# B&R Automation Studio project DivDiag (part 2)

### DivertRepo.mpreportcore - PC/mappServices/DivertRepo.mpreportcore
```
Element gOffsetsReport (Type=mpreportcore)
  MpReport:
    Settings:
      ResourceDeviceName = 
      LanguageDependent:
        [0]:
          Language = en
          Font = 1
    PageLayouts:
      [0]:
        Name = Default
        PageFormat = 1
    Styles:
      Text:
        [0]:
          Name = Default
        [1]:
          Name = Title
          Style = 1
          Size = 14
        [2]:
          Name = Header
          Size = 12
        [3]:
          Name = Section
          Style = 2
          Size = 12
      Table:
        [0]:
          Name = Default
      Line:
        [0]:
          Name = Default
      Chart:
        PieChart:
          [0]:
            Name = Default
        LineChart:
          [0]:
            Name = Default
        BarChart:
          [0]:
            Name = Default
    Tables:
      [0]:
        Name = Divert1
        TableStyle = Default
        TextStyle = Default
        [0]:
          [0] = TextId
            Source = 
            Width = 40
          [1] = TextId
            Source = Segment 1
          [2] = TextId
            Source = Segment 2
        [1]:
          [0] = TextId
            Source = Name
            Width = 40
          [1] = ValueId
            Value:
              ProcessVariable = ::Maint:TestResults[0].Seg1Name
          [2] = ValueId
            Value:
              ProcessVariable = ::Maint:TestResults[0].Seg2Name
        [2]:
          [0] = TextId
            Source = Type
            Width = 40
          [1] = ValueId
            Value:
              ProcessVariable = ::Maint:TestResults[0].Seg1Type
          [2] = ValueId
            Value:
              ProcessVariable = ::Maint:TestResults[0].Seg2Type
        [3]:
          [0] = TextId
            Source = Relative to start of segment
            Width = 40
          [1] = ValueId
            Value:
              ProcessVariable = ::Maint:TestResults[0].Seg1PosRelToStart
          [2] = ValueId
            Value:
              ProcessVariable = ::Maint:TestResults[0].Seg2PosRelToStart
        [4]:
          [0] = TextId
            Source = Relative to end of segment
            Width = 40
          [1] = ValueId
            Value:
              ProcessVariable = ::Maint:TestResults[0].Seg1PosRelToEnd
          [2] = ValueId
            Value:
              ProcessVariable = ::Maint:TestResults[0].Seg2PosRelToEnd
        [5]:
          [0] = TextId
            Source = Measured Configuration Mismatch
            Width = 40
          [1] = ValueId
            Value:
              ProcessVariable = ::Maint:TestResults[0].Deviation
            Width = 50
            HorizontalAlign = 1
      [1]:
        Name = Divert2
        TableStyle = Default
        TextStyle = Default
        [0]:
          [0] = TextId
            Source = 
            Width = 40
          [1] = TextId
            Source = Segment 1
          [2] = TextId
            Source = Segment 2
        [1]:
          [0] = TextId
            Source = Name
            Width = 40
          [1] = ValueId
            Value:
              ProcessVariable = ::Maint:TestResults[1].Seg1Name
          [2] = ValueId
            Value:
              ProcessVariable = ::Maint:TestResults[1].Seg2Name
        [2]:
          [0] = TextId
            Source = Type
            Width = 40
          [1] = ValueId
            Value:
              ProcessVariable = ::Maint:TestResults[1].Seg1Type
          [2] = ValueId
            Value:
              ProcessVariable = ::Maint:TestResults[1].Seg2Type
        [3]:
          [0] = TextId
            Source = Relative to start of segment
            Width = 40
          [1] = ValueId
            Value:
              ProcessVariable = ::Maint:TestResults[1].Seg1PosRelToStart
          [2] = ValueId
            Value:
              ProcessVariable = ::Maint:TestResults[1].Seg2PosRelToStart
        [4]:
          [0] = TextId
            Source = Relative to end of segment
            Width = 40
          [1] = ValueId
            Value:
              ProcessVariable = ::Maint:TestResults[1].Seg1PosRelToEnd
          [2] = ValueId
            Value:
              ProcessVariable = ::Maint:TestResults[1].Seg2PosRelToEnd
        [5]:
          [0] = TextId
            Source = Measured Configuration Mismatch
            Width = 40
          [1] = ValueId
            Value:
              ProcessVariable = ::Maint:TestResults[1].Deviation
            Width = 50
            HorizontalAlign = 1
      [2]:
        Name = Divert3
        TableStyle = Default
        TextStyle = Default
        [0]:
          [0] = TextId
            Source = 
            Width = 40
          [1] = TextId
            Source = Segment 1
          [2] = TextId
            Source = Segment 2
        [1]:
          [0] = TextId
            Source = Name
            Width = 40
          [1] = ValueId
            Value:
              ProcessVariable = ::Maint:TestResults[2].Seg1Name
          [2] = ValueId
            Value:
              ProcessVariable = ::Maint:TestResults[2].Seg2Name
        [2]:
          [0] = TextId
            Source = Type
            Width = 40
          [1] = ValueId
            Value:
              ProcessVariable = ::Maint:TestResults[2].Seg1Type
          [2] = ValueId
            Value:
              ProcessVariable = ::Maint:TestResults[2].Seg2Type
        [3]:
          [0] = TextId
            Source = Relative to start of segment
            Width = 40
          [1] = ValueId
            Value:
              ProcessVariable = ::Maint:TestResults[2].Seg1PosRelToStart
          [2] = ValueId
            Value:
              ProcessVariable = ::Maint:TestResults[2].Seg2PosRelToStart
        [4]:
          [0] = TextId
            Source = Relative to end of segment
            Width = 40
          [1] = ValueId
            Value:
              ProcessVariable = ::Maint:TestResults[2].Seg1PosRelToEnd
          [2] = ValueId
            Value:
              ProcessVariable = ::Maint:TestResults[2].Seg2PosRelToEnd
        [5]:
          [0] = TextId
            Source = Measured Configuration Mismatch
            Width = 40
          [1] = ValueId
            Value:
              ProcessVariable = ::Maint:TestResults[2].Deviation
            Width = 50
            HorizontalAlign = 1
      [3]:
        Name = Divert4
        TableStyle = Default
        TextStyle = Default
        [0]:
          [0] = TextId
            Source = 
            Width = 40
          [1] = TextId
            Source = Segment 1
          [2] = TextId
            Source = Segment 2
        [1]:
          [0] = TextId
            Source = Name
            Width = 40
          [1] = ValueId
            Value:
              ProcessVariable = ::Maint:TestResults[3].Seg1Name
          [2] = ValueId
            Value:
              ProcessVariable = ::Maint:TestResults[3].Seg2Name
        [2]:
          [0] = TextId
            Source = Type
            Width = 40
          [1] = ValueId
            Value:
              ProcessVariable = ::Maint:TestResults[3].Seg1Type
          [2] = ValueId
            Value:
              ProcessVariable = ::Maint:TestResults[3].Seg2Type
        [3]:
          [0] = TextId
            Source = Relative to start of segment
            Width = 40
          [1] = ValueId
            Value:
              ProcessVariable = ::Maint:TestResults[3].Seg1PosRelToStart
          [2] = ValueId
            Value:
              ProcessVariable = ::Maint:TestResults[3].Seg2PosRelToStart
        [4]:
          [0] = TextId
            Source = Relative to end of segment
            Width = 40
          [1] = ValueId
            Value:
              ProcessVariable = ::Maint:TestResults[3].Seg1PosRelToEnd
          [2] = ValueId
            Value:
              ProcessVariable = ::Maint:TestResults[3].Seg2PosRelToEnd
        [5]:
          [0] = TextId
            Source = Measured Configuration Mismatch
            Width = 40
          [1] = ValueId
            Value:
              ProcessVariable = ::Maint:TestResults[3].Deviation
            Width = 50
            HorizontalAlign = 1
      [4]:
        Name = Divert5
        TableStyle = Default
        TextStyle = Default
        [0]:
          [0] = TextId
            Source = 
            Width = 40
          [1] = TextId
            Source = Segment 1
          [2] = TextId
            Source = Segment 2
        [1]:
          [0] = TextId
            Source = Name
            Width = 40
          [1] = ValueId
            Value:
              ProcessVariable = ::Maint:TestResults[4].Seg1Name
          [2] = ValueId
            Value:
              ProcessVariable = ::Maint:TestResults[4].Seg2Name
        [2]:
          [0] = TextId
            Source = Type
            Width = 40
          [1] = ValueId
            Value:
              ProcessVariable = ::Maint:TestResults[4].Seg1Type
          [2] = ValueId
            Value:
              ProcessVariable = ::Maint:TestResults[4].Seg2Type
        [3]:
          [0] = TextId
            Source = Relative to start of segment
            Width = 40
          [1] = ValueId
            Value:
              ProcessVariable = ::Maint:TestResults[4].Seg1PosRelToStart
          [2] = ValueId
            Value:
              ProcessVariable = ::Maint:TestResults[4].Seg2PosRelToStart
        [4]:
          [0] = TextId
            Source = Relative to end of segment
            Width = 40
          [1] = ValueId
            Value:
              ProcessVariable = ::Maint:TestResults[4].Seg1PosRelToEnd
          [2] = ValueId
            Value:
              ProcessVariable = ::Maint:TestResults[4].Seg2PosRelToEnd
        [5]:
          [0] = TextId
            Source = Measured Configuration Mismatch
            Width = 40
          [1] = ValueId
            Value:
              ProcessVariable = ::Maint:TestResults[4].Deviation
            Width = 50
            HorizontalAlign = 1
      [5]:
        Name = Divert6
        TableStyle = Default
        TextStyle = Default
        [0]:
          [0] = TextId
            Source = 
            Width = 40
          [1] = TextId
            Source = Segment 1
          [2] = TextId
            Source = Segment 2
        [1]:
          [0] = TextId
            Source = Name
            Width = 40
          [1] = ValueId
            Value:
              ProcessVariable = ::Maint:TestResults[5].Seg1Name
          [2] = ValueId
            Value:
              ProcessVariable = ::Maint:TestResults[5].Seg2Name
        [2]:
          [0] = TextId
            Source = Type
            Width = 40
          [1] = ValueId
            Value:
              ProcessVariable = ::Maint:TestResults[5].Seg1Type
          [2] = ValueId
            Value:
              ProcessVariable = ::Maint:TestResults[5].Seg2Type
        [3]:
          [0] = TextId
            Source = Relative to start of segment
            Width = 40
          [1] = ValueId
            Value:
              ProcessVariable = ::Maint:TestResults[5].Seg1PosRelToStart
          [2] = ValueId
            Value:
              ProcessVariable = ::Maint:TestResults[5].Seg2PosRelToStart
        [4]:
          [0] = TextId
            Source = Relative to end of segment
            Width = 40
          [1] = ValueId
            Value:
              ProcessVariable = ::Maint:TestResults[5].Seg1PosRelToEnd
          [2] = ValueId
            Value:
              ProcessVariable = ::Maint:TestResults[5].Seg2PosRelToEnd
        [5]:
          [0] = TextId
            Source = Measured Configuration Mismatch
            Width = 40
          [1] = ValueId
            Value:
              ProcessVariable = ::Maint:TestResults[5].Deviation
            Width = 50
            HorizontalAlign = 1
      [6]:
        Name = Divert7
        TableStyle = Default
        TextStyle = Default
        [0]:
          [0] = TextId
            Source = 
            Width = 40
          [1] = TextId
            Source = Segment 1
          [2] = TextId
            Source = Segment 2
        [1]:
          [0] = TextId
            Source = Name
            Width = 40
          [1] = ValueId
            Value:
              ProcessVariable = ::Maint:TestResults[6].Seg1Name
          [2] = ValueId
            Value:
              ProcessVariable = ::Maint:TestResults[6].Seg2Name
        [2]:
          [0] = TextId
            Source = Type
            Width = 40
          [1] = ValueId
            Value:
              ProcessVariable = ::Maint:TestResults[6].Seg1Type
          [2] = ValueId
            Value:
              ProcessVariable = ::Maint:TestResults[6].Seg2Type
        [3]:
          [0] = TextId
            Source = Relative to start of segment
            Width = 40
          [1] = ValueId
            Value:
              ProcessVariable = ::Maint:TestResults[6].Seg1PosRelToStart
          [2] = ValueId
            Value:
              ProcessVariable = ::Maint:TestResults[6].Seg2PosRelToStart
        [4]:
          [0] = TextId
            Source = Relative to end of segment
            Width = 40
          [1] = ValueId
            Value:
              ProcessVariable = ::Maint:TestResults[6].Seg1PosRelToEnd
          [2] = ValueId
            Value:
              ProcessVariable = ::Maint:TestResults[6].Seg2PosRelToEnd
        [5]:
          [0] = TextId
            Source = Measured Configuration Mismatch
            Width = 40
          [1] = ValueId
            Value:
              ProcessVariable = ::Maint:TestResults[6].Deviation
            Width = 50
            HorizontalAlign = 1
      [7]:
        Name = Divert8
        TableStyle = Default
        TextStyle = Default
        [0]:
          [0] = TextId
            Source = 
            Width = 40
          [1] = TextId
            Source = Segment 1
          [2] = TextId
            Source = Segment 2
        [1]:
          [0] = TextId
            Source = Name
            Width = 40
          [1] = ValueId
            Value:
              ProcessVariable = ::Maint:TestResults[7].Seg1Name
          [2] = ValueId
            Value:
              ProcessVariable = ::Maint:TestResults[7].Seg2Name
        [2]:
          [0] = TextId
            Source = Type
            Width = 40
          [1] = ValueId
            Value:
              ProcessVariable = ::Maint:TestResults[7].Seg1Type
          [2] = ValueId
            Value:
              ProcessVariable = ::Maint:TestResults[7].Seg2Type
        [3]:
          [0] = TextId
            Source = Relative to start of segment
            Width = 40
          [1] = ValueId
            Value:
              ProcessVariable = ::Maint:TestResults[7].Seg1PosRelToStart
          [2] = ValueId
            Value:
              ProcessVariable = ::Maint:TestResults[7].Seg2PosRelToStart
        [4]:
          [0] = TextId
            Source = Relative to end of segment
            Width = 40
          [1] = ValueId
            Value:
              ProcessVariable = ::Maint:TestResults[7].Seg1PosRelToEnd
          [2] = ValueId
            Value:
              ProcessVariable = ::Maint:TestResults[7].Seg2PosRelToEnd
        [5]:
          [0] = TextId
            Source = Measured Configuration Mismatch
            Width = 40
          [1] = ValueId
            Value:
              ProcessVariable = ::Maint:TestResults[7].Deviation
            Width = 50
            HorizontalAlign = 1
      [8]:
        Name = Divert9
        TableStyle = Default
        TextStyle = Default
        [0]:
          [0] = TextId
            Source = 
            Width = 40
          [1] = TextId
            Source = Segment 1
          [2] = TextId
            Source = Segment 2
        [1]:
          [0] = TextId
            Source = Name
            Width = 40
          [1] = ValueId
            Value:
              ProcessVariable = ::Maint:TestResults[8].Seg1Name
          [2] = ValueId
            Value:
              ProcessVariable = ::Maint:TestResults[8].Seg2Name
        [2]:
          [0] = TextId
            Source = Type
            Width = 40
          [1] = ValueId
            Value:
              ProcessVariable = ::Maint:TestResults[8].Seg1Type
          [2] = ValueId
            Value:
              ProcessVariable = ::Maint:TestResults[8].Seg2Type
        [3]:
          [0] = TextId
            Source = Relative to start of segment
            Width = 40
          [1] = ValueId
            Value:
              ProcessVariable = ::Maint:TestResults[8].Seg1PosRelToStart
          [2] = ValueId
            Value:
              ProcessVariable = ::Maint:TestResults[8].Seg2PosRelToStart
        [4]:
          [0] = TextId
            Source = Relative to end of segment
            Width = 40
          [1] = ValueId
            Value:
              ProcessVariable = ::Maint:TestResults[8].Seg1PosRelToEnd
          [2] = ValueId
            Value:
              ProcessVariable = ::Maint:TestResults[8].Seg2PosRelToEnd
        [5]:
          [0] = TextId
            Source = Measured Configuration Mismatch
            Width = 40
          [1] = ValueId
            Value:
              ProcessVariable = ::Maint:TestResults[8].Deviation
            Width = 50
            HorizontalAlign = 1
      [9]:
        Name = Divert10
        TableStyle = Default
        TextStyle = Default
        [0]:
          [0] = TextId
            Source = 
            Width = 40
          [1] = TextId
            Source = Segment 1
          [2] = TextId
            Source = Segment 2
        [1]:
          [0] = TextId
            Source = Name
            Width = 40
          [1] = ValueId
            Value:
              ProcessVariable = ::Maint:TestResults[9].Seg1Name
          [2] = ValueId
            Value:
              ProcessVariable = ::Maint:TestResults[9].Seg2Name
        [2]:
          [0] = TextId
            Source = Type
            Width = 40
          [1] = ValueId
            Value:
              ProcessVariable = ::Maint:TestResults[9].Seg1Type
          [2] = ValueId
            Value:
              ProcessVariable = ::Maint:TestResults[9].Seg2Type
        [3]:
          [0] = TextId
            Source = Relative to start of segment
            Width = 40
          [1] = ValueId
            Value:
              ProcessVariable = ::Maint:TestResults[9].Seg1PosRelToStart
          [2] = ValueId
            Value:
              ProcessVariable = ::Maint:TestResults[9].Seg2PosRelToStart
        [4]:
          [0] = TextId
            Source = Relative to end of segment
            Width = 40
          [1] = ValueId
            Value:
              ProcessVariable = ::Maint:TestResults[9].Seg1PosRelToEnd
          [2] = ValueId
            Value:
              ProcessVariable = ::Maint:TestResults[9].Seg2PosRelToEnd
        [5]:
          [0] = TextId
            Source = Measured Configuration Mismatch
            Width = 40
          [1] = ValueId
            Value:
              ProcessVariable = ::Maint:TestResults[9].Deviation
            Width = 50
            HorizontalAlign = 1
      [10]:
        Name = Divert11
        TableStyle = Default
        TextStyle = Default
        [0]:
          [0] = TextId
            Source = 
            Width = 40
          [1] = TextId
            Source = Segment 1
          [2] = TextId
            Source = Segment 2
        [1]:
          [0] = TextId
            Source = Name
            Width = 40
          [1] = ValueId
            Value:
              ProcessVariable = ::Maint:TestResults[10].Seg1Name
          [2] = ValueId
            Value:
              ProcessVariable = ::Maint:TestResults[10].Seg2Name
        [2]:
          [0] = TextId
            Source = Type
            Width = 40
          [1] = ValueId
            Value:
              ProcessVariable = ::Maint:TestResults[10].Seg1Type
          [2] = ValueId
            Value:
              ProcessVariable = ::Maint:TestResults[10].Seg2Type
        [3]:
          [0] = TextId
            Source = Relative to start of segment
            Width = 40
          [1] = ValueId
            Value:
              ProcessVariable = ::Maint:TestResults[10].Seg1PosRelToStart
          [2] = ValueId
            Value:
              ProcessVariable = ::Maint:TestResults[10].Seg2PosRelToStart
        [4]:
          [0] = TextId
            Source = Relative to end of segment
            Width = 40
          [1] = ValueId
            Value:
              ProcessVariable = ::Maint:TestResults[10].Seg1PosRelToEnd
          [2] = ValueId
            Value:
              ProcessVariable = ::Maint:TestResults[10].Seg2PosRelToEnd
        [5]:
          [0] = TextId
            Source = Measured Configuration Mismatch
            Width = 40
          [1] = ValueId
            Value:
              ProcessVariable = ::Maint:TestResults[10].Deviation
            Width = 50
            HorizontalAlign = 1
      [11]:
        Name = Divert12
        TableStyle = Default
        TextStyle = Default
        [0]:
          [0] = TextId
            Source = 
            Width = 40
          [1] = TextId
            Source = Segment 1
          [2] = TextId
            Source = Segment 2
        [1]:
          [0] = TextId
            Source = Name
            Width = 40
          [1] = ValueId
            Value:
              ProcessVariable = ::Maint:TestResults[11].Seg1Name
          [2] = ValueId
            Value:
              ProcessVariable = ::Maint:TestResults[11].Seg2Name
        [2]:
          [0] = TextId
            Source = Type
            Width = 40
          [1] = ValueId
            Value:
              ProcessVariable = ::Maint:TestResults[11].Seg1Type
          [2] = ValueId
            Value:
              ProcessVariable = ::Maint:TestResults[11].Seg2Type
        [3]:
          [0] = TextId
            Source = Relative to start of segment
            Width = 40
          [1] = ValueId
            Value:
              ProcessVariable = ::Maint:TestResults[11].Seg1PosRelToStart
          [2] = ValueId
            Value:
              ProcessVariable = ::Maint:TestResults[11].Seg2PosRelToStart
        [4]:
          [0] = TextId
            Source = Relative to end of segment
            Width = 40
          [1] = ValueId
            Value:
              ProcessVariable = ::Maint:TestResults[11].Seg1PosRelToEnd
          [2] = ValueId
            Value:
              ProcessVariable = ::Maint:TestResults[11].Seg2PosRelToEnd
        [5]:
          [0] = TextId
            Source = Measured Configuration Mismatch
            Width = 40
          [1] = ValueId
            Value:
              ProcessVariable = ::Maint:TestResults[11].Deviation
            Width = 50
            HorizontalAlign = 1
    Charts:
      [0] = BarChart
        Name = DeviationBarChart
        Heading = SingleText
          Text = Diverter Offset Mismatch Measurements
          HorizontalAlign = 1
          TextStyle = Section
        ChartStyle = Default
        TextStyle = Default
        ShowLegend = 2
        YAxis:
          Label = Deviation (m)
          NumberOfGridLines = 4
          ItemMinValue = Dynamic
            ValuePV = ::Maint:MinDeviation
          ItemMaxValue = Dynamic
            ValuePV = ::Maint:MaxDeviation
        [0]:
          Value:
            ProcessVariable = ::Maint:TestResults[0].Deviation
          LegendText = Diverter 1
        [1]:
          Value:
            ProcessVariable = ::Maint:TestResults[1].Deviation
          ItemColor = FF0000
          LegendText = Diverter 2
        [2]:
          Value:
            ProcessVariable = ::Maint:TestResults[2].Deviation
          ItemColor = 7F7F7F
          LegendText = Diverter 3
        [3]:
          Value:
            ProcessVariable = ::Maint:TestResults[3].Deviation
          ItemColor = 800000
          LegendText = Diverter 4
        [4]:
          Value:
            ProcessVariable = ::Maint:TestResults[4].Deviation
          ItemColor = FFFF00
          LegendText = Diverter 5
        [5]:
          Value:
            ProcessVariable = ::Maint:TestResults[5].Deviation
          ItemColor = 800080
          LegendText = Diverter 6
        [6]:
          Value:
            ProcessVariable = ::Maint:TestResults[6].Deviation
          ItemColor = 00FFFF
          LegendText = Diverter 7
        [7]:
          Value:
            ProcessVariable = ::Maint:TestResults[7].Deviation
          ItemColor = 33CC00
          LegendText = Diverter 8
        [8]:
          Value:
            ProcessVariable = ::Maint:TestResults[8].Deviation
          ItemColor = FF9900
          LegendText = Diverter 9
        [9]:
          Value:
            ProcessVariable = ::Maint:TestResults[9].Deviation
          ItemColor = 808000
          LegendText = Diverter 10
        [10]:
          Value:
            ProcessVariable = ::Maint:TestResults[10].Deviation
          LegendText = Diverter 11
        [11]:
          Value:
            ProcessVariable = ::Maint:TestResults[11].Deviation
          ItemColor = FF0000
          LegendText = Diverter 12
    Contents:
      [0]:
        Name = Header
        [0]:
          Text = Diverter Offset Results
          HorizontalAlign = 1
          NewLine = FALSE
          TextStyle = Title
        [1] = EmptyLine
          Size = 16
        [2]:
          Text = gMcAssembly01
          NewLine = FALSE
          TextStyle = Header
        [3] = DateTime
          HorizontalAlign = 2
          NewLine = FALSE
          TextStyle = Header
        [4] = EmptyLine
          Size = 14
      [1]:
        Name = Diverter1
        [0] = Table
          Table = Divert1
          HorizontalAlign = 1
        [1] = EmptyLine
          Size = 16
      [2]:
        Name = Diverter2
        [0] = Table
          Table = Divert2
          HorizontalAlign = 1
        [1] = EmptyLine
          Size = 16
      [3]:
        Name = Diverter3
        [0] = Table
          Table = Divert3
          HorizontalAlign = 1
        [1] = EmptyLine
          Size = 16
      [4]:
        Name = Diverter4
        [0] = Table
          Table = Divert4
          HorizontalAlign = 1
        [1] = EmptyLine
          Size = 16
      [5]:
        Name = Diverter5
        [0] = Table
          Table = Divert5
          HorizontalAlign = 1
        [1] = EmptyLine
          Size = 16
      [6]:
        Name = Diverter6
        [0] = Table
          Table = Divert6
          HorizontalAlign = 1
        [1] = EmptyLine
          Size = 16
      [7]:
        Name = Diverter7
        [0] = Table
          Table = Divert7
          HorizontalAlign = 1
        [1] = EmptyLine
          Size = 16
      [8]:
        Name = Diverter8
        [0] = Table
          Table = Divert8
          HorizontalAlign = 1
        [1] = EmptyLine
          Size = 16
      [9]:
        Name = Diverter9
        [0] = Table
          Table = Divert9
          HorizontalAlign = 1
        [1] = EmptyLine
          Size = 16
      [10]:
        Name = Diverter10
        [0] = Table
          Table = Divert10
          HorizontalAlign = 1
        [1] = EmptyLine
          Size = 16
      [11]:
        Name = Diverter11
        [0] = Table
          Table = Divert11
          HorizontalAlign = 1
        [1] = EmptyLine
          Size = 16
      [12]:
        Name = Diverter12
        [0] = Table
          Table = Divert12
          HorizontalAlign = 1
        [1] = EmptyLine
          Size = 16
      [13]:
        Name = Chart
        [0] = Chart
          Chart = DeviationBarChart
          HorizontalAlign = 1
    Reports:
      [0]:
        Name = DiverterOffsetResults
        Settings:
          AllowCopy = TRUE
        FileNamePattern = DiverterOffsets_%Y_%m_%d_%H_%M_%S.pdf
        PageLayout = Default
        Header = Header
        [0]:
          Heading:
            Text = Diverter 1
            TextStyle = Section
          [0]:
            Content = Diverter1
        [1]:
          Heading:
            Text = Diverter 2
            TextStyle = Section
          [0]:
            Content = Diverter2
        [2]:
          Heading:
            Text = Diverter 3
            TextStyle = Section
          [0]:
            Content = Diverter3
        [3]:
          Heading:
            Text = Diverter 4
            TextStyle = Section
          [0]:
            Content = Diverter4
        [4]:
          Heading:
            Text = Diverter 5
            TextStyle = Section
          [0]:
            Content = Diverter5
        [5]:
          Heading:
            Text = Diverter 6
            TextStyle = Section
          [0]:
            Content = Diverter6
        [6]:
          Heading:
            Text = Diverter 7
            TextStyle = Section
          [0]:
            Content = Diverter7
        [7]:
          Heading:
            Text = Diverter 8
            TextStyle = Section
          [0]:
            Content = Diverter8
        [8]:
          Heading:
            Text = Diverter 9
            TextStyle = Section
          [0]:
            Content = Diverter9
        [9]:
          Heading:
            Text = Diverter 10
            TextStyle = Section
          [0]:
            Content = Diverter10
        [10]:
          Heading:
            Text = Diverter 11
            TextStyle = Section
          [0]:
            Content = Diverter11
        [11]:
          Heading:
            Text = Diverter 12
            TextStyle = Section
          [0]:
            Content = Diverter12
        [12]:
          StartOnNewPage = TRUE
          Heading:
            TextStyle = Section
          [0]:
            Content = Chart
```

## Configuration PCSim

### Task classes (Cpu.sw)
```
Libraries: CoTrace, AsZip, FileIO, runtime
```

### Hardware
```
5LS182.6-2 : 5LS182.6-2 v1.7.1.0  [SL -> PC.SL1]
  Connector IF1:
    CycleTime = 800
PC : PC_any v1.1.1.0 (OrderNumber=PC)
  ConfigurationID = DivDiag_PCSim
  SystemTick = 800
  FileDevice1
  FileDeviceName1 = SvgData
  FileDevicePath1 = ../../../Scene/Generated
  FtpUser1
  FtpUsername1 = user  // user
  FtpUserPassword1 = jyjjSNMo3acQF/SzeDpvbTiMzVTrFM+cM4mnOTaTPJ4=  // user
  FtpUserSalt1 = 14QPuDID
  FTPAccessRight1 = 0
  ActivateOpcUa = 1
  OpcUaInformationModels_PV_Version = 1
```

## Logical view

Binary libraries used (declarations not repeated): operator, runtime, astime, AsIecCon, McBase, CoTrace, AsZip, FileIO, McAcpTrak, McAxis, standard, AsBrStr, McAcpPar, sys_lib, AsIODiag

### Package Logical/Libraries - Global libraries

### SourceGlobal.var - Segments Definition
```iecst
VAR
	gSysIf : SysIfTyp;
END_VAR
```

### SourceGlobal.typ - Global data types
```iecst
TYPE
	SysStateEnum :
		(
		SYS_OFF,
		SYS_POWERING_ON,
		SYS_POWERING_OFF,
		SYS_ADD_SHUTTLE,
		SYS_IDLE,
		SYS_ERROR
		);
	SysIfTyp : 	STRUCT
		Cmd : SysIfCmdTyp;
		Sts : SysIfStsTyp;
	END_STRUCT;
	SysIfCmdTyp : 	STRUCT
		PowerOn : BOOL;
	END_STRUCT;
	SysIfStsTyp : 	STRUCT
		Powered : BOOL;
		ShuttleAdded : BOOL;
	END_STRUCT;
	SysFbsTyp : 	STRUCT
		AsmPowerFb : MC_BR_AsmPowerOn_AcpTrak;
		AsmPowerOffFb : MC_BR_AsmPowerOff_AcpTrak;
		AddShuttleFb : MC_BR_SecAddShuttle_AcpTrak;
	END_STRUCT;
END_TYPE
```

### Segments.var - Segments Definition
```iecst
(*MC objects - Main loop*)
VAR
	SEG_A_10 : McSegmentType;
	SEG_A_11 : McSegmentType;
	SEG_A_12 : McSegmentType;
	SEG_A_13 : McSegmentType;
	SEG_A_14 : McSegmentType;
	SEG_A_15 : McSegmentType;
	SEG_A_16 : McSegmentType;
	SEG_A_17 : McSegmentType;
	SEG_A_18 : McSegmentType;
	SEG_A_19 : McSegmentType;
	SEG_A_20 : McSegmentType;
	SEG_A_21 : McSegmentType;
	SEG_A_22 : McSegmentType;
	SEG_A_23 : McSegmentType;
	SEG_A_24 : McSegmentType;
	SEG_A_25 : McSegmentType;
	SEG_A_26 : McSegmentType;
	SEG_A_27 : McSegmentType;
	SEG_A_28 : McSegmentType;
	SEG_A_29 : McSegmentType;
	SEG_A_30 : McSegmentType;
	SEG_A_31 : McSegmentType;
	SEG_A_32 : McSegmentType;
	SEG_A_33 : McSegmentType;
	SEG_A_34 : McSegmentType;
	SEG_A_35 : McSegmentType;
	SEG_A_36 : McSegmentType;
	SEG_A_37 : McSegmentType;
	SEG_A_38 : McSegmentType;
	SEG_A_39 : McSegmentType;
	SEG_A_40 : McSegmentType;
	SEG_A_41 : McSegmentType;
	SEG_A_42 : McSegmentType;
	SEG_A_43 : McSegmentType;
	SEG_A_44 : McSegmentType;
	SEG_A_45 : McSegmentType;
	SEG_A_46 : McSegmentType;
	SEG_A_47 : McSegmentType;
	SEG_A_48 : McSegmentType;
	SEG_A_49 : McSegmentType;
	SEG_A_50 : McSegmentType;
END_VAR
(**)
(*MC objects - B Track QC loop*)
VAR
	SEG_B_40 : McSegmentType;
	SEG_B_41 : McSegmentType;
	SEG_B_42 : McSegmentType;
	SEG_B_43 : McSegmentType;
	SEG_B_44 : McSegmentType;
	SEG_B_45 : McSegmentType;
	SEG_B_46 : McSegmentType;
	SEG_B_47 : McSegmentType;
	SEG_B_48 : McSegmentType;
	SEG_B_49 : McSegmentType;
	SEG_B_50 : McSegmentType;
	SEG_B_51 : McSegmentType;
	SEG_B_52 : McSegmentType;
	SEG_B_53 : McSegmentType;
	SEG_B_54 : McSegmentType;
	SEG_B_55 : McSegmentType;
	SEG_B_56 : McSegmentType;
	SEG_B_57 : McSegmentType;
END_VAR
(**)
(*MC objects - C Track*)
VAR
	SEG_C_20 : McSegmentType;
	SEG_C_21 : McSegmentType;
	SEG_C_22 : McSegmentType;
	SEG_C_23 : McSegmentType;
	SEG_C_24 : McSegmentType;
	SEG_C_25 : McSegmentType;
	SEG_C_26 : McSegmentType;
	SEG_C_27 : McSegmentType;
	SEG_C_28 : McSegmentType;
	SEG_C_29 : McSegmentType;
	SEG_C_30 : McSegmentType;
	SEG_C_31 : McSegmentType;
END_VAR
(**)
(*MC objects - D Track*)
VAR
	SEG_D_10 : McSegmentType;
	SEG_D_11 : McSegmentType;
	SEG_D_12 : McSegmentType;
	SEG_D_13 : McSegmentType;
	SEG_D_14 : McSegmentType;
	SEG_D_15 : McSegmentType;
	SEG_D_16 : McSegmentType;
	SEG_D_32 : McSegmentType;
	SEG_D_33 : McSegmentType;
	SEG_D_34 : McSegmentType;
	SEG_D_35 : McSegmentType;
	SEG_D_36 : McSegmentType;
	SEG_D_37 : McSegmentType;
	SEG_D_38 : McSegmentType;
END_VAR
(**)
(*MC objects - Flex track #1 *)
VAR
	SEG_E_13 : McSegmentType;
	SEG_E_14 : McSegmentType;
	SEG_E_15 : McSegmentType;
	SEG_E_16 : McSegmentType;
	SEG_E_17 : McSegmentType;
	SEG_E_18 : McSegmentType;
	SEG_E_19 : McSegmentType;
	SEG_E_20 : McSegmentType;
	SEG_E_21 : McSegmentType;
	SEG_E_22 : McSegmentType;
	SEG_E_23 : McSegmentType;
	SEG_E_24 : McSegmentType;
	SEG_E_25 : McSegmentType;
	SEG_E_26 : McSegmentType;
	SEG_E_60 : McSegmentType;
	SEG_E_61 : McSegmentType;
END_VAR
(**)
(*MC objects - Flex #1 OUT*)
VAR
	SEG_F_27 : McSegmentType;
	SEG_F_28 : McSegmentType;
	SEG_F_29 : McSegmentType;
	SEG_F_30 : McSegmentType;
	SEG_F_31 : McSegmentType;
	SEG_F_32 : McSegmentType;
	SEG_F_33 : McSegmentType;
	SEG_F_34 : McSegmentType;
	SEG_F_35 : McSegmentType;
	SEG_F_70 : McSegmentType;
	SEG_F_71 : McSegmentType;
END_VAR
(**)
(*MC objects - Flex #2 IN*)
VAR
	SEG_G_10 : McSegmentType;
	SEG_G_11 : McSegmentType;
	SEG_G_12 : McSegmentType;
	SEG_G_13 : McSegmentType;
	SEG_G_14 : McSegmentType;
	SEG_G_15 : McSegmentType;
	SEG_G_16 : McSegmentType;
	SEG_G_17 : McSegmentType;
	SEG_G_18 : McSegmentType;
	SEG_G_19 : McSegmentType;
END_VAR
(**)
(*MC objects - Flex track #2 *)
VAR
	SEG_H_10 : McSegmentType;
	SEG_H_11 : McSegmentType;
	SEG_H_12 : McSegmentType;
	SEG_H_13 : McSegmentType;
	SEG_H_14 : McSegmentType;
	SEG_H_15 : McSegmentType;
	SEG_H_16 : McSegmentType;
	SEG_H_17 : McSegmentType;
	SEG_H_18 : McSegmentType;
	SEG_H_19 : McSegmentType;
	SEG_H_20 : McSegmentType;
	SEG_H_21 : McSegmentType;
	SEG_H_22 : McSegmentType;
	SEG_H_23 : McSegmentType;
	SEG_H_24 : McSegmentType;
	SEG_H_25 : McSegmentType;
	SEG_H_26 : McSegmentType;
	SEG_H_27 : McSegmentType;
END_VAR
(**)
(*MC objects - Flex #2 OUT*)
VAR
	SEG_I_30 : McSegmentType;
	SEG_I_31 : McSegmentType;
	SEG_I_32 : McSegmentType;
	SEG_I_33 : McSegmentType;
	SEG_I_34 : McSegmentType;
	SEG_I_35 : McSegmentType;
END_VAR
(**)
(*MC objects - X-ray #1*)
VAR
	SEG_J_35 : McSegmentType;
	SEG_J_36 : McSegmentType;
	SEG_J_37 : McSegmentType;
	SEG_J_38 : McSegmentType;
	SEG_J_39 : McSegmentType;
	SEG_J_40 : McSegmentType;
	SEG_J_41 : McSegmentType;
	SEG_J_42 : McSegmentType;
END_VAR
(**)
(*MC objects - X-ray #2*)
VAR
	SEG_K_35 : McSegmentType;
	SEG_K_36 : McSegmentType;
	SEG_K_37 : McSegmentType;
	SEG_K_38 : McSegmentType;
	SEG_K_39 : McSegmentType;
	SEG_K_40 : McSegmentType;
	SEG_K_41 : McSegmentType;
	SEG_K_42 : McSegmentType;
END_VAR
(**)
(*MC objects - Track L*)
VAR
	SEG_L_50 : McSegmentType;
END_VAR
(**)
(*MC objects - Track M*)
VAR
	SEG_M_60 : McSegmentType;
	SEG_M_61 : McSegmentType;
	SEG_M_62 : McSegmentType;
	SEG_M_63 : McSegmentType;
	SEG_M_64 : McSegmentType;
	SEG_M_65 : McSegmentType;
	SEG_M_66 : McSegmentType;
	SEG_M_67 : McSegmentType;
	SEG_M_68 : McSegmentType;
	SEG_M_69 : McSegmentType;
	SEG_M_70 : McSegmentType;
	SEG_M_71 : McSegmentType;
	SEG_M_72 : McSegmentType;
END_VAR
```

### Program Logical/Source/MainTest (IEC)

#### Variables.var
```iecst
VAR
	state : SysStateEnum;
	sysFbs : SysFbsTyp;
END_VAR
```

#### Cyclic.st
```iecst
PROGRAM _CYCLIC
	CASE state OF
		SYS_OFF:
			IF gSysIf.Cmd.PowerOn THEN
				sysFbs.AsmPowerFb.Assembly := ADR(gMcAssembly01);
				sysFbs.AsmPowerFb.Execute := TRUE;
				state := SYS_POWERING_ON;
			END_IF
		SYS_POWERING_ON:
			IF sysFbs.AsmPowerFb.Done THEN
				gSysIf.Sts.Powered := TRUE;

				IF gSysIf.Sts.ShuttleAdded THEN
					state := SYS_IDLE;
				ELSE
					sysFbs.AddShuttleFb.Position := 0;
					sysFbs.AddShuttleFb.Sector := ADR(gDivSector_0);
					sysFbs.AddShuttleFb.Execute := TRUE;

					state := SYS_ADD_SHUTTLE;
				END_IF
			END_IF
		SYS_POWERING_OFF:
			IF sysFbs.AsmPowerOffFb.Done THEN
				sysFbs.AsmPowerOffFb.Execute := FALSE;
				gSysIf.Sts.Powered := FALSE;
				state := SYS_OFF;
			END_IF
		SYS_ADD_SHUTTLE:
			IF sysFbs.AddShuttleFb.Error THEN
				state := SYS_ERROR;
			ELSIF sysFbs.AddShuttleFb.Done THEN
				sysFbs.AddShuttleFb.Execute := FALSE;
				gSysIf.Sts.ShuttleAdded := TRUE;

				state := SYS_IDLE;
			END_IF
		SYS_IDLE:
			IF NOT gSysIf.Cmd.PowerOn THEN
				sysFbs.AsmPowerOffFb.Execute := TRUE;
				sysFbs.AsmPowerOffFb.Assembly := ADR(gMcAssembly01);

				state := SYS_POWERING_OFF;
			END_IF
		SYS_ERROR:

	END_CASE;

	sysFbs.AsmPowerFb();
	sysFbs.AsmPowerOffFb();
	sysFbs.AddShuttleFb();

END_PROGRAM
```

### Program Logical/Source/Diagnostic/Maint (IEC) - Maintenance Program

#### Cyclic.st - Cyclic code
```iecst
PROGRAM _CYCLIC

	IF DivertTestOffsets.Done THEN
	    DivertTestOffsets.Execute := 0;
	    brsmemcpy(ADR(TestResults), ADR(DivertTestOffsets.Config), SIZEOF(TestResults));
	    FOR i := 0 TO mlMAX_DIVERT_IDX DO
	        IF i = 0 THEN
	            MaxDeviation := TestResults[i].Deviation;
	            MinDeviation := TestResults[i].Deviation;
	        ELSE
	            MaxDeviation := MAX(MaxDeviation, TestResults[i].Deviation);
	            MinDeviation := MIN(MinDeviation, TestResults[i].Deviation);
	        END_IF
	    END_FOR

	END_IF

	DivertTestOffsets();

END_PROGRAM
```

#### Init.st - Init code
```iecst
//This file was automatically generated using the Diverter Diagnostic program. Verify that the segment names and assembly name match your project values correctly
PROGRAM _INIT
	DivertTestOffsets.Sectors[0] := gDivSector_0;	//SEG_D_10:TrackSegmentType.AB SegmentRelativeTo.FromStart at 0.0 connected to SEG_A_39:TrackSegmentType.AA SegmentRelativeTo.FromEnd at 0.000621 type DivReferenceType.RelToOne
	DivertTestOffsets.Sectors[1] := gDivSector_1;	//SEG_E_16:TrackSegmentType.AA SegmentRelativeTo.FromEnd at 0.0 connected to SEG_D_15:TrackSegmentType.AA SegmentRelativeTo.FromEnd at 0.104015 type DivReferenceType.RelToOne
	//DivertTestOffsets.Sectors[2] := gDivSector_2;	//SEG_F_30:TrackSegmentType.AA SegmentRelativeTo.FromStart at 0.0 connected to SEG_E_24:TrackSegmentType.AA SegmentRelativeTo.FromStart at 0.0 type DivReferenceType.RelToTwo
	//DivertTestOffsets.Sectors[3] := gDivSector_3;	//SEG_F_35:TrackSegmentType.BA SegmentRelativeTo.FromStart at 0.0 connected to SEG_A_35:TrackSegmentType.AA SegmentRelativeTo.FromStart at 0.0 type DivReferenceType.RelToTwo
	DivertTestOffsets.Sectors[4] := gDivSector_4;	//SEG_J_42:TrackSegmentType.AB SegmentRelativeTo.FromStart at 0.0 connected to SEG_D_13:TrackSegmentType.AA SegmentRelativeTo.FromStart at 0.254651 type DivReferenceType.RelToOne
	DivertTestOffsets.Sectors[5] := gDivSector_5;	//SEG_H_16:TrackSegmentType.AA SegmentRelativeTo.FromEnd at 0.0 connected to SEG_G_15:TrackSegmentType.AA SegmentRelativeTo.FromEnd at 0.106253 type DivReferenceType.RelToOne
	//DivertTestOffsets.Sectors[6] := gDivSector_6;	//SEG_I_30:TrackSegmentType.AA SegmentRelativeTo.FromStart at 0.0 connected to SEG_H_24:TrackSegmentType.AA SegmentRelativeTo.FromStart at 0.0 type DivReferenceType.RelToTwo
	//DivertTestOffsets.Sectors[7] := gDivSector_7;	//SEG_I_35:TrackSegmentType.BA SegmentRelativeTo.FromStart at 0.0 connected to SEG_A_30:TrackSegmentType.AA SegmentRelativeTo.FromStart at 0.0 type DivReferenceType.RelToTwo
	DivertTestOffsets.Sectors[8] := gDivSector_8;	//SEG_K_42:TrackSegmentType.AB SegmentRelativeTo.FromStart at 0 connected to SEG_G_13:TrackSegmentType.AA SegmentRelativeTo.FromStart at 0.25575255 type DivReferenceType.RelToOne
	DivertTestOffsets.ShSourceSector := ADR(gDivSector_0);
	DivertTestOffsets.SegmentName1[0] := 'SEG_D_10';
	DivertTestOffsets.SegmentName2[0] := 'SEG_A_39';
	DivertTestOffsetsPar.Positions[0] := 0.045;
	DivertTestOffsets.SegmentName1[1] := 'SEG_E_16';
	DivertTestOffsets.SegmentName2[1] := 'SEG_D_15';
	DivertTestOffsetsPar.Positions[1] := 0.045;
	DivertTestOffsets.SegmentName1[2] := 'SEG_F_30';
	DivertTestOffsets.SegmentName2[2] := 'SEG_E_24';
	DivertTestOffsetsPar.Positions[2] := 0.045;
	DivertTestOffsets.SegmentName1[3] := 'SEG_F_35';
	DivertTestOffsets.SegmentName2[3] := 'SEG_A_35';
	DivertTestOffsetsPar.Positions[3] := 0.045;
	DivertTestOffsets.SegmentName1[4] := 'SEG_J_42';
	DivertTestOffsets.SegmentName2[4] := 'SEG_D_13';
	DivertTestOffsetsPar.Positions[4] := 0.045;
	DivertTestOffsets.SegmentName1[5] := 'SEG_H_16';
	DivertTestOffsets.SegmentName2[5] := 'SEG_G_15';
	DivertTestOffsetsPar.Positions[5] := 0.045;
	DivertTestOffsets.SegmentName1[6] := 'SEG_I_30';
	DivertTestOffsets.SegmentName2[6] := 'SEG_H_24';
	DivertTestOffsetsPar.Positions[6] := 0.045;
	DivertTestOffsets.SegmentName1[7] := 'SEG_I_35';
	DivertTestOffsets.SegmentName2[7] := 'SEG_A_30';
	DivertTestOffsetsPar.Positions[7] := 0.045;
	DivertTestOffsets.SegmentName1[8] := 'SEG_K_42';
	DivertTestOffsets.SegmentName2[8] := 'SEG_G_13';
	DivertTestOffsetsPar.Positions[8] := 0.045;

	DivertTestOffsets.Parameters := ADR(DivertTestOffsetsPar);
	DivertTestOffsetsPar.Velocity := 1.0;
	DivertTestOffsetsPar.Acceleration := 20.0;
	DivertTestOffsetsPar.Deceleration := 20.0;
	DivertTestOffsetsPar.SettleTime := T#5s;
END_PROGRAM
```

#### Types.typ - Local data types
```iecst
TYPE
	StateEnum :
		( (*State of execution*)
		STATE_IDLE, (*Wait for teach command*)
		STATE_MAINTENANCE_INIT, (*Initialize maintenance*)
		STATE_CLEAR_UPSTREAM, (*Clear upstream*)
		STATE_CLEAR_DOWNSTREAM, (*Clear downstream*)
		STATE_CLEAR_ALL, (*Clear all*)
		STATE_SEND_RETURN, (*Send shuttles to the return*)
		STATE_GET_OFFSET, (*Get divert offset commanded*)
		STATE_TEST_OFFSETS, (*Test diverter offsets*)
		STATE_DONE (*Maintenance command is complete*)
		);
END_TYPE
```

#### Variables.var - Local variables
```iecst
VAR
	State : StateEnum; (*State of execution*)
	GetSegOffset : GetSegmentOffsets; (*Get segment offset*)
	DivertTestOffsets : TestOffsets; (*Test assembly divert offsets*)
	DivertTestOffsetsPar : TestOffsetsParType; (*Divert offset test parameters*)
	TestResults : ARRAY[0..mlMAX_DIVERT_IDX] OF GetSegmentOffsetsConfigType; (*Test results from divert test*)
	MaxDeviation : REAL; (*Maximum Diverter Deviation*)
	MinDeviation : REAL; (*Minimum Diverter Deviation*)
	i : USINT; (*Index*)
END_VAR
(*Constants*)
VAR CONSTANT
	ERR_NO_SH_ON_SEC : DINT := -10000; (*No shuttles found on sector*)
	ERR_INVALID_SEG_TYPE : DINT := -10001; (*The segment type is invalid*)
	ERR_INVALID_CONFIG : DINT := -10002; (*Resulting configuration is invalid*)
	mlMAX_DIVERT_IDX : USINT := 20;
END_VAR
```

#### FunctionTypes.typ - Local function types
```iecst
(*Get Segment Offsets*)

TYPE
	GetSegmentOffsetsConfigType : 	STRUCT  (*Configuration result*)
		Seg1Name : STRING[32]; (*Segment 1 name*)
		Seg2Name : STRING[32]; (*Segment 2 name*)
		Seg1Type : STRING[80]; (*track segment 1 type*)
		Seg2Type : STRING[80]; (*segment 2 type*)
		Deviation : REAL; (*result CmdCheckConfigDeviation:
measured deviation of diverter segment mounting to assembly-track-configuration [m]*)
		Seg1PosRelToStart : REAL; (*result CmdCheckConfigDeviation:
suggested value to enter in assembly-track-configuration for  track segment 1 "Position" if "Position relative to = Start of segment" [m]*)
		Seg1PosRelToEnd : REAL; (*result CmdCheckConfigDeviation:
suggested value to enter in assembly-track-configuration for track segment 1 "Position" if "Position relative to = End of segment" [m]*)
		Seg2PosRelToStart : REAL; (*result CmdCheckConfigDeviation:
suggested value to enter in assembly-track-configuration for track segment 2 "Position" if "Position relative to = Start of segment" [m]*)
		Seg2PosRelToEnd : REAL; (*result CmdCheckConfigDeviation:
suggested value to enter in assembly-track-configuration for  track segment 2 "Position" if "Position relative to = End of segment" [m]*)
	END_STRUCT;
	GetSegmentOffsetsInternalType : 	STRUCT  (*Internal Data*)
		State : GetSegmentOffsetsStateEnum; (*State of execution*)
		Status1 : DINT; (*Return status 1*)
		Status2 : DINT; (*Return status 2*)
		Seg1Ref : UDINT; (*Segment 1 reference*)
		Seg1Len : UDINT; (*Segment 1 data length*)
		Seg2Ref : UDINT; (*Segment 2 reference*)
		Seg2Len : UDINT; (*Segment 2 data length*)
		ProductCode1 : UDINT; (*Segment 1 read product code*)
		ProductCode2 : UDINT; (*Segment 2 read product code*)
		PosAct1 : DINT; (*Segment 1 read actual position*)
		PosAct2 : DINT; (*Segment 2 read actual position*)
		Position1 : REAL; (*Position on the segment*)
		Position2 : REAL; (*Position on the segment*)
		LagError1 : REAL; (*Segment 1 read lag error*)
		LagError2 : REAL; (*Segment 2 read lag error*)
		SegProcessParID1 : MC_BR_SegProcessParID_AcpTrak; (*Process segment 1 parameters*)
		ParId1 : ARRAY[0..2]OF McAcpTrakSegProcessParIDType; (*Segment 1 parameters*)
		SegProcessParID2 : MC_BR_SegProcessParID_AcpTrak; (*Process segment 2 parameters*)
		ParId2 : ARRAY[0..2]OF McAcpTrakSegProcessParIDType; (*Segment 2 parameters*)
		SegType1 : GetSegType; (*Get segment 1 type*)
		SegType2 : GetSegType; (*Get segment 2 type*)
	END_STRUCT;
	GetSegmentOffsetsStateEnum :
		( (*State of execution*)
		GET_OFFSET_STATE_IDLE, (*Idle state*)
		GET_OFFSET_STATE_GET_SEG, (*Get segment addresses from PV names*)
		GET_OFFSET_STATE_GET_VALUES, (*Get values from segments*)
		GET_OFFSET_STATE_GET_TYPE, (*Get segment type*)
		GET_OFFSET_STATE_DONE, (*Offsets found*)
		GET_OFFSET_STATE_RESET_FB, (*Reset function blocks*)
		GET_OFFSET_STATE_WAIT_NOT_BUSY, (*Wait for function blocks to report not busy*)
		GET_OFFSET_STATE_ERROR (*An error occurred*)
		);
END_TYPE

(*Send To Return*)

TYPE
	SendToReturnParType : 	STRUCT  (*Parameters*)
		SendDelay : TIME; (*Time to wait between sending shuttles*)
		CheckInterval : TIME; (*Time to wait between checking for completion*)
		PosRelativeTo : McAcpTrakRoutePosRelToEnum; (*Whether the position is relative to the start or end of the sector*)
		Position : LREAL; (*Position to send shuttles to*)
		Velocity : REAL; (*Move velocity*)
		Acceleration : REAL; (*Move acceleration*)
		Deceleration : REAL; (*Move deceleration*)
	END_STRUCT;
	SendToReturnInternalType : 	STRUCT  (*Internal Data*)
		State : SendToReturnStateEnum; (*State of execution*)
		AsmGetShuttle : MC_BR_AsmGetShuttle_AcpTrak; (*Get shuttles on the assembly*)
		RoutedMoveAbs : MC_BR_RoutedMoveAbs_AcpTrak; (*Send shuttles with a routed move absolute*)
		ShReadInfo : MC_BR_ShReadInfo_AcpTrak; (*Read shuttle information*)
		DelayTON : TON; (*Delay sending the next shuttle*)
		CheckTON : TON; (*Wait to check for completion*)
		OldRemainingCount : UDINT; (*Previously recorded value of the remaining count*)
	END_STRUCT;
	SendToReturnStateEnum :
		( (*State of execution*)
		SEND_RETURN_STATE_IDLE, (*Idle state*)
		SEND_RETURN_STATE_GET_SH_SEND, (*Get shuttles for sending*)
		SEND_RETURN_STATE_SEND_SH, (*Send shuttle*)
		SEND_RETURN_STATE_DELAY, (*Delay sending the next shuttle*)
		SEND_RETURN_STATE_NEXT_SH_SEND, (*Get next shuttle for sending*)
		SEND_RETURN_STATE_WAIT_CHECK, (*Wait to check for shuttle move done*)
		SEND_RETURN_STATE_GET_SH_CHECK, (*Get shuttles for checking for completion*)
		SEND_RETURN_STATE_SH_INFO, (*Check if shuttle is stopped*)
		SEND_RETURN_STATE_NEXT_SH_CHECK, (*Get the next shuttle to check*)
		SEND_RETURN_STATE_DONE, (*All shuttles are on the return*)
		SEND_RETURN_STATE_RESET_FB, (*Reset function blocks*)
		SEND_RETURN_STATE_WAIT_NOT_BUSY, (*Wait for function blocks to report not busy*)
		SEND_RETURN_STATE_ERROR (*An error occurred*)
		);
END_TYPE

(*Test Offsets*)

TYPE
	TestOffsetsParType : 	STRUCT  (*Parameters*)
		Positions : ARRAY[0..mlMAX_DIVERT_IDX]OF LREAL; (*Positions on each divert sector*)
		PosRelativeTo : ARRAY[0..mlMAX_DIVERT_IDX]OF McAcpTrakRoutePosRelToEnum; (*Whether the position is relative to the start or end of the sector*)
		Velocity : REAL; (*Move velocity*)
		Acceleration : REAL; (*Move acceleration*)
		Deceleration : REAL; (*Move deceleration*)
		SettleTime : TIME; (*Time to wait before measuring position*)
	END_STRUCT;
	TestOffsetsInternalType : 	STRUCT  (*Internal Data*)
		State : TestOffsetsStateEnum; (*State of execution*)
		SecGetShuttle : MC_BR_SecGetShuttle_AcpTrak; (*Get shuttle for test*)
		RoutedMoveAbs : MC_BR_RoutedMoveAbs_AcpTrak; (*Send shuttle*)
		GetSegOffsets : GetSegmentOffsets; (*Get segment offsets*)
		SettleTON : TON; (*Timer*)
		DivertIndex : USINT; (*Current Divert index*)
	END_STRUCT;
	TestOffsetsStateEnum :
		( (*State of execution*)
		TEST_OFFSETS_STATE_IDLE, (*Idle state*)
		TEST_OFFSETS_STATE_GET_SH, (*Get shuttle*)
		TEST_OFFSETS_STATE_SEND, (*Send shuttle*)
		TEST_OFFSETS_STATE_SETTLE, (*Wait for settling*)
		TEST_OFFSETS_STATE_GET_SEG, (*Get segments*)
		TEST_OFFSETS_STATE_DONE, (*Testing complete*)
		TEST_OFFSETS_STATE_RESET_FB, (*Reset function blocks*)
		TEST_OFFSETS_STATE_WAIT_NOT_BUSY, (*Wait for function blocks to report not busy*)
		TEST_OFFSETS_STATE_ERROR (*An error occurred*)
		);
END_TYPE
```

#### LocalFunctions.fun - Local functions
```iecst
FUNCTION_BLOCK GetSegmentOffsets (*Get segment offsets*)
	VAR_INPUT
		SegmentName1 : STRING[32]; (*Name of the first divert segment*)
		SegmentName2 : STRING[32]; (*Name of the second divert segment*)
		Execute : BOOL; (*Get offsets of the selected segments*)
	END_VAR
	VAR_OUTPUT
		Busy : BOOL; (*The function block is busy and must continue to be called*)
		Done : BOOL; (*The data has been captured*)
		Config : GetSegmentOffsetsConfigType; (*Suggested configuration*)
		Error : BOOL; (*An error occurred*)
		ErrorID : DINT; (*ID of the error that occurred*)
	END_VAR
	VAR
		Internal : GetSegmentOffsetsInternalType; (*Internal Data*)
	END_VAR
END_FUNCTION_BLOCK

FUNCTION_BLOCK TestOffsets (*Test Segment offsets*)
	VAR_INPUT
		ShSourceSector : REFERENCE TO McSectorType; (*Shuttle to pull from for test*)
		Parameters : REFERENCE TO TestOffsetsParType; (*Parameters*)
		SegmentName1 : ARRAY[0..mlMAX_DIVERT_IDX] OF STRING[32]; (*Name of the first divert segment*)
		SegmentName2 : ARRAY[0..mlMAX_DIVERT_IDX] OF STRING[32]; (*Name of the second divert segment*)
		Sectors : ARRAY[0..mlMAX_DIVERT_IDX] OF McSectorType; (*Sectors to use for sending to the divert*)
		Execute : BOOL; (*Test offsets*)
	END_VAR
	VAR_OUTPUT
		Busy : BOOL; (*The function block is busy and must continue to be called*)
		Done : BOOL; (*The data has been captured*)
		Config : ARRAY[0..mlMAX_DIVERT_IDX] OF GetSegmentOffsetsConfigType; (*Test results*)
		Error : BOOL; (*An error occurred*)
		ErrorID : DINT; (*ID of the error that occurred*)
	END_VAR
	VAR
		Internal : TestOffsetsInternalType; (*Internal Data*)
	END_VAR
END_FUNCTION_BLOCK

FUNCTION_BLOCK GetSegType (*Return data about the segment type*)
	VAR_INPUT
		ProductCode : UDINT; (*Segment product code*)
		Execute : BOOL; (*Return segment data*)
	END_VAR
	VAR_OUTPUT
		Valid : BOOL; (*If true, the output is valid*)
		Error : BOOL; (*An error occurred*)
		ErrorID : DINT; (*ID of the error that occurred*)
		Type : STRING[80]; (*Segment type*)
		Length : REAL; (*Segment length*)
	END_VAR
END_FUNCTION_BLOCK
```

#### GetSegmentOffsets.st - Get offset between two segments
```iecst
(* Get segment offset data *)
FUNCTION_BLOCK GetSegmentOffsets

    CASE Internal.State OF

        GET_OFFSET_STATE_IDLE:

            IF Execute THEN
                Busy := 1;
                Internal.ParId1[0].ParID := mcACPPAR_EPROM_PRODUCT_CODE;
                Internal.ParId1[0].DataType := mcACPTRAK_SEG_PARTYPE_UDINT;
                Internal.ParId1[0].VariableAddress := ADR(Internal.ProductCode1);
                Internal.ParId1[1].ParID := mcACPPAR_ENCOD0_POS_ACT;
                Internal.ParId1[1].DataType := mcACPTRAK_SEG_PARTYPE_DINT;
                Internal.ParId1[1].VariableAddress := ADR(Internal.PosAct1);
                Internal.ParId1[2].ParID := mcACPPAR_PCTRL_LAG_ERROR;
                Internal.ParId1[2].DataType := mcACPTRAK_SEG_PARTYPE_REAL;
                Internal.ParId1[2].VariableAddress := ADR(Internal.LagError1);
                Internal.ParId2[0].ParID := mcACPPAR_EPROM_PRODUCT_CODE;
                Internal.ParId2[0].DataType := mcACPTRAK_SEG_PARTYPE_UDINT;
                Internal.ParId2[0].VariableAddress := ADR(Internal.ProductCode2);
                Internal.ParId2[1].ParID := mcACPPAR_ENCOD0_POS_ACT;
                Internal.ParId2[1].DataType := mcACPTRAK_SEG_PARTYPE_DINT;
                Internal.ParId2[1].VariableAddress := ADR(Internal.PosAct2);
                Internal.ParId2[2].ParID := mcACPPAR_PCTRL_LAG_ERROR;
                Internal.ParId2[2].DataType := mcACPTRAK_SEG_PARTYPE_REAL;
                Internal.ParId2[2].VariableAddress := ADR(Internal.LagError2);
                Internal.SegProcessParID1.DataAddress := ADR(Internal.ParId1);
                Internal.SegProcessParID1.NumberOfParIDs := 3;
                Internal.SegProcessParID1.Mode := mcACPTRAK_SEG_PARID_GET;
                Internal.SegProcessParID1.ChannelIndex := 0;
                Internal.SegProcessParID2.DataAddress := ADR(Internal.ParId2);
                Internal.SegProcessParID2.NumberOfParIDs := 3;
                Internal.SegProcessParID2.Mode := mcACPTRAK_SEG_PARID_GET;
                Internal.SegProcessParID2.ChannelIndex := 0;
                Internal.Status1 := PV_xgetadr(ADR(SegmentName1), ADR(Internal.Seg1Ref), ADR(Internal.Seg1Len));
                Internal.Status2 := PV_xgetadr(ADR(SegmentName2), ADR(Internal.Seg2Ref), ADR(Internal.Seg2Len));

				Internal.State := GET_OFFSET_STATE_DONE;
				//Internal.State := GET_OFFSET_STATE_GET_SEG;
            END_IF

        GET_OFFSET_STATE_GET_SEG:

            IF Internal.Status1 <> ERR_OK THEN
                Error := 1;
                ErrorID := Internal.Status1;
                Internal.State := GET_OFFSET_STATE_RESET_FB;
            ELSIF Internal.Status2 <> ERR_OK THEN
                Error := 1;
                ErrorID := Internal.Status2;
                Internal.State := GET_OFFSET_STATE_RESET_FB;
            ELSE
                Internal.SegProcessParID1.Segment := Internal.Seg1Ref;
                Internal.SegProcessParID2.Segment := Internal.Seg2Ref;
                Internal.SegProcessParID1.Execute := 1;
                Internal.SegProcessParID2.Execute := 1;
                Internal.State := GET_OFFSET_STATE_GET_VALUES;
            END_IF

        GET_OFFSET_STATE_GET_VALUES:

            IF Internal.SegProcessParID1.Error THEN
                Error := 1;
                ErrorID := Internal.SegProcessParID1.ErrorID;
                Internal.State := GET_OFFSET_STATE_RESET_FB;
            ELSIF Internal.SegProcessParID2.Error THEN
                Error := 1;
                ErrorID := Internal.SegProcessParID2.ErrorID;
                Internal.State := GET_OFFSET_STATE_RESET_FB;
            ELSIF Internal.SegProcessParID1.Done AND Internal.SegProcessParID2.Done THEN
                Internal.SegProcessParID1.Execute := 0;
                Internal.SegProcessParID2.Execute := 0;
                Internal.Position1 := DINT_TO_REAL(Internal.PosAct1)/10000000.0;
                Internal.Position2 := DINT_TO_REAL(Internal.PosAct2)/10000000.0;
                Internal.SegType1.ProductCode := Internal.ProductCode1;
                Internal.SegType1.Execute := 1;
                Internal.SegType2.ProductCode := Internal.ProductCode2;
                Internal.SegType2.Execute := 1;
                Internal.State := GET_OFFSET_STATE_GET_TYPE;
            END_IF

        GET_OFFSET_STATE_GET_TYPE:

            IF Internal.SegType1.Error THEN
                Error := 1;
                ErrorID := Internal.SegType1.ErrorID;
                Internal.State := GET_OFFSET_STATE_RESET_FB;
            ELSIF Internal.SegType2.Error THEN
                Error := 1;
                ErrorID := Internal.SegType2.ErrorID;
                Internal.State := GET_OFFSET_STATE_RESET_FB;
            ELSIF Internal.SegType1.Valid AND Internal.SegType2.Valid THEN
                Internal.SegType1.Execute := 0;
                Internal.SegType2.Execute := 0;
                // calculate track-connection point at the pos/neg end of track segment 2
                IF(Internal.Position2 <= (Internal.SegType2.Length/2.0))THEN
                    Config.Seg2PosRelToStart	:= 0.0;
                    Config.Seg2PosRelToEnd	    := Internal.SegType2.Length;
                    Config.Seg1PosRelToStart	:= Internal.Position1 + Internal.Position2;
                ELSE
                    Config.Seg2PosRelToStart	:= Internal.SegType2.Length;
                    Config.Seg2PosRelToEnd	    := 0.0;
                    Config.Seg1PosRelToStart	:= Internal.Position1 - (Internal.SegType2.Length - Internal.Position2);
                END_IF
                Config.Seg1PosRelToEnd		    := Internal.SegType1.Length - Config.Seg1PosRelToStart;
                Config.Deviation	            := Internal.LagError1 + Internal.LagError2;

                // shift track-connection point if it is outside the existing track segment
                IF(Config.Seg1PosRelToStart < 0.0)THEN
                    Config.Seg2PosRelToStart	:= Config.Seg2PosRelToStart	+ Config.Seg1PosRelToStart;
                    Config.Seg2PosRelToEnd	    := Config.Seg2PosRelToEnd	- Config.Seg1PosRelToStart;
                    Config.Seg1PosRelToStart	:= 0.0;
                    Config.Seg1PosRelToEnd	    := Internal.SegType1.Length;
                END_IF
                IF(Config.Seg1PosRelToEnd < 0.0)THEN
                    Config.Seg2PosRelToStart	:= Config.Seg2PosRelToStart	- Config.Seg1PosRelToEnd;
                    Config.Seg2PosRelToEnd	    := Config.Seg2PosRelToEnd	+ Config.Seg1PosRelToEnd;
                    Config.Seg1PosRelToStart	:= Internal.SegType1.Length;
                    Config.Seg1PosRelToEnd	    := 0.0;
                END_IF

                // check for result valid
                IF(	(Internal.SegType1.Length > 0.0) AND
                    (Internal.Position1 <> 0.0) AND
                    (Config.Seg1PosRelToStart >= 0.0) AND
                    (Config.Seg1PosRelToStart <= Internal.SegType1.Length) AND
                    (Config.Seg1PosRelToEnd >= 0.0) AND
                    (Config.Seg1PosRelToEnd <= Internal.SegType1.Length) AND
                    (Internal.SegType2.Length > 0.0) AND
                    (Internal.Position2 <> 0.0) AND
                    (Config.Seg2PosRelToStart >= 0.0) AND
                    (Config.Seg2PosRelToStart <= Internal.SegType2.Length) AND
                    (Config.Seg2PosRelToEnd >= 0.0) AND
                    (Config.Seg2PosRelToEnd <= Internal.SegType2.Length) )THEN
                    brsstrcpy(ADR(Config.Seg1Name), ADR(SegmentName1));
                    brsstrcpy(ADR(Config.Seg2Name), ADR(SegmentName2));
                    brsstrcpy(ADR(Config.Seg1Type), ADR(Internal.SegType1.Type));
                    brsstrcpy(ADR(Config.Seg2Type), ADR(Internal.SegType2.Type));
                    Done := 1;
                    Internal.State := GET_OFFSET_STATE_DONE;
                ELSE
                    Error := 1;
                    ErrorID := ERR_INVALID_CONFIG;
                    Internal.State := GET_OFFSET_STATE_RESET_FB;
                END_IF
            END_IF

        GET_OFFSET_STATE_DONE:

            IF NOT Execute THEN
                Done := 0;
                brsmemset(ADR(Config), 0, SIZEOF(Config));
                Internal.State := GET_OFFSET_STATE_WAIT_NOT_BUSY;
            END_IF

        GET_OFFSET_STATE_RESET_FB:

            Internal.SegProcessParID1.Execute := 0;
            Internal.SegProcessParID2.Execute := 0;
            Internal.SegType1.Execute := 0;
            Internal.SegType2.Execute := 0;
            IF Error THEN
                Internal.State := GET_OFFSET_STATE_ERROR;
            ELSE
                Internal.State := GET_OFFSET_STATE_WAIT_NOT_BUSY;
            END_IF

        GET_OFFSET_STATE_WAIT_NOT_BUSY:

            IF NOT (Internal.SegProcessParID1.Busy OR Internal.SegProcessParID2.Busy) THEN
                Busy := 0;
                Internal.State := GET_OFFSET_STATE_IDLE;
            END_IF

        GET_OFFSET_STATE_ERROR:

            IF NOT Execute THEN
                Error := 0;
                ErrorID := ERR_OK;
                Internal.State := GET_OFFSET_STATE_WAIT_NOT_BUSY;
            END_IF

    END_CASE

    Internal.SegProcessParID1();
    Internal.SegProcessParID2();
    Internal.SegType1();
    Internal.SegType2();

END_FUNCTION_BLOCK
```

#### TestOffsets.st - Test segment offsets
```iecst
FUNCTION_BLOCK TestOffsets

    CASE Internal.State OF

        TEST_OFFSETS_STATE_IDLE:

            IF Execute THEN
                Busy := TRUE;
                Internal.DivertIndex := FALSE;
                Internal.SecGetShuttle.Sector := ADR(ShSourceSector);
                Internal.SecGetShuttle.Mode := mcACPTRAK_SEARCH_BACKWARD;
                Internal.SecGetShuttle.Enable := TRUE;
                Internal.RoutedMoveAbs.Axis := ADR(Internal.SecGetShuttle.Axis);
                Internal.RoutedMoveAbs.Velocity := Parameters.Velocity;
                Internal.RoutedMoveAbs.Acceleration := Parameters.Acceleration;
                Internal.RoutedMoveAbs.Deceleration := Parameters.Deceleration;
                Internal.RoutedMoveAbs.AdvancedParameters.StartDirection := mcDIR_UNDEFINED;
                Internal.RoutedMoveAbs.AdvancedParameters.EndDirection := mcDIR_POSITIVE;
                Internal.RoutedMoveAbs.AdvancedParameters.ShuttleOrientation := mcDIR_UNDEFINED;
                Internal.SettleTON.PT := Parameters.SettleTime;
                Internal.State := TEST_OFFSETS_STATE_GET_SH;
            END_IF

        TEST_OFFSETS_STATE_GET_SH:

            IF NOT Execute THEN
                Internal.State := TEST_OFFSETS_STATE_RESET_FB;
            ELSIF Internal.SecGetShuttle.Error THEN
                Error := TRUE;
                ErrorID := Internal.SecGetShuttle.ErrorID;
                Internal.State := TEST_OFFSETS_STATE_RESET_FB;
            ELSIF Internal.SecGetShuttle.Valid THEN
                IF Internal.SecGetShuttle.TotalCount = 0 THEN
                    Error := TRUE;
                    ErrorID := ERR_NO_SH_ON_SEC;
                    Internal.State := TEST_OFFSETS_STATE_RESET_FB;
                ELSE
                    Internal.RoutedMoveAbs.Sector := ADR(Sectors[Internal.DivertIndex]);
                    Internal.RoutedMoveAbs.Position := Parameters.Positions[Internal.DivertIndex];
                    Internal.RoutedMoveAbs.AdvancedParameters.PosRelativeTo := Parameters.PosRelativeTo[Internal.DivertIndex];
                    Internal.RoutedMoveAbs.Execute := TRUE;
                    Internal.State := TEST_OFFSETS_STATE_SEND;
                END_IF
            END_IF

        TEST_OFFSETS_STATE_SEND:

            IF NOT Execute THEN
                Internal.State := TEST_OFFSETS_STATE_RESET_FB;
            ELSIF Internal.RoutedMoveAbs.Error THEN
                Error := TRUE;
                ErrorID := Internal.RoutedMoveAbs.ErrorID;
                Internal.State := TEST_OFFSETS_STATE_RESET_FB;
            ELSIF Internal.RoutedMoveAbs.Done THEN
                Internal.RoutedMoveAbs.Execute := FALSE;
                Internal.SettleTON.IN := TRUE;
                Internal.State := TEST_OFFSETS_STATE_SETTLE;
            END_IF

        TEST_OFFSETS_STATE_SETTLE:

            IF NOT Execute THEN
                Internal.State := TEST_OFFSETS_STATE_RESET_FB;
            ELSIF Internal.SettleTON.Q THEN
                Internal.SettleTON.IN := FALSE;
                Internal.GetSegOffsets.SegmentName1 := SegmentName1[Internal.DivertIndex];
                Internal.GetSegOffsets.SegmentName2 := SegmentName2[Internal.DivertIndex];
                Internal.GetSegOffsets.Execute:= TRUE;
                Internal.State := TEST_OFFSETS_STATE_GET_SEG;
            END_IF

        TEST_OFFSETS_STATE_GET_SEG:

            IF NOT Execute THEN
                Internal.State := TEST_OFFSETS_STATE_RESET_FB;
            ELSIF Internal.GetSegOffsets.Error THEN
                Error := TRUE;
                ErrorID := Internal.GetSegOffsets.ErrorID;
                Internal.State := TEST_OFFSETS_STATE_RESET_FB;
            ELSIF Internal.GetSegOffsets.Done THEN
                Internal.GetSegOffsets.Execute := FALSE;
                brsmemcpy(ADR(Config[Internal.DivertIndex]), ADR(Internal.GetSegOffsets.Config), SIZEOF(Config[Internal.DivertIndex]));
                IF Internal.DivertIndex < mlMAX_DIVERT_IDX THEN
                    Internal.DivertIndex := Internal.DivertIndex + TRUE;
                    Internal.RoutedMoveAbs.Sector := ADR(Sectors[Internal.DivertIndex]);
                    Internal.RoutedMoveAbs.Position := Parameters.Positions[Internal.DivertIndex];
                    Internal.RoutedMoveAbs.AdvancedParameters.PosRelativeTo := Parameters.PosRelativeTo[Internal.DivertIndex];
                    Internal.RoutedMoveAbs.Execute := TRUE;
                    Internal.State := TEST_OFFSETS_STATE_SEND;
                ELSE
                    Internal.SecGetShuttle.Enable := FALSE;
                    Done := TRUE;
                    Internal.State := TEST_OFFSETS_STATE_DONE;
                END_IF
            END_IF

        TEST_OFFSETS_STATE_DONE:

            IF NOT Execute THEN
                Done := FALSE;
                brsmemset(ADR(Config), 0, SIZEOF(Config));
                Internal.State := TEST_OFFSETS_STATE_WAIT_NOT_BUSY;
            END_IF

        TEST_OFFSETS_STATE_RESET_FB:

            Internal.SecGetShuttle.Enable := FALSE;
            Internal.RoutedMoveAbs.Execute := FALSE;
            Internal.GetSegOffsets.Execute := FALSE;
            Internal.SettleTON.IN := FALSE;
            IF Error THEN
                Internal.State := TEST_OFFSETS_STATE_ERROR;
            ELSE
                Internal.State := TEST_OFFSETS_STATE_WAIT_NOT_BUSY;
            END_IF

        TEST_OFFSETS_STATE_WAIT_NOT_BUSY:

            IF NOT (Internal.SecGetShuttle.Busy OR Internal.RoutedMoveAbs.Busy OR Internal.GetSegOffsets.Busy) THEN
                Busy := FALSE;
                Internal.State := TEST_OFFSETS_STATE_IDLE;
            END_IF

        TEST_OFFSETS_STATE_ERROR:

            IF NOT Execute THEN
                Error := FALSE;
                ErrorID := ERR_OK;
                Internal.State := TEST_OFFSETS_STATE_WAIT_NOT_BUSY;
            END_IF

    END_CASE

    Internal.SecGetShuttle();
    Internal.RoutedMoveAbs();
    Internal.GetSegOffsets();
    Internal.SettleTON();

END_FUNCTION_BLOCK
```

#### GetSegType.st - Get segment type
```iecst
FUNCTION_BLOCK GetSegType

    IF Execute THEN
        CASE ProductCode OF
            16#EBFE:
                Type	:= 'PT1 8YFIZ1.AA63.00-1';
                Length	:= 0.630;
                Valid := 1;
            16#EE0A:
                Type	:= 'PT1 8YFIZ1.AA63.10-1';
                Length	:= 0.630;
                Valid := 1;
            16#EC00:
                Type	:= 'PT1 8YFIZ1.AB43.00-1';
                Length	:= 0.435642;
                Valid := 1;
            16#EE0B:
                Type	:= 'PT1 8YFIZ1.AB43.10-1';
                Length	:= 0.435642;
                Valid := 1;
            16#EC01:
                Type	:= 'PT1 8YFIZ1.BA43.00-1';
                Length	:= 0.435642;
                Valid := 1;
            16#EE0C:
                Type	:= 'PT1 8YFIZ1.BA43.10-1';
                Length	:= 0.435642;
                Valid := 1;
            16#F255:
                Type	:= 'PT2 8YF1I01.AA66.00-1';
                Length	:= 0.660;
                Valid := 1;
            16#F256:
                Type	:= 'PT2 8YF1I01.AB2B.00-1';
                Length	:= 0.450585;
                Valid := 1;
            16#F257:
                Type	:= 'PT2 8YF1I01.BA2B.00-1';
                Length	:= 0.450585;
                Valid := 1;
            16#F7C3:
                Type	:= '8F1I01.AA66.0000-1';
                Length	:= 0.660;
                Valid := 1;
            16#F7CA:
                Type	:= '8F1I01.BB4B.0000-1 invalid for diverter!';
                Length	:= 0.240;
                Error := 1;
                ErrorID := ERR_INVALID_SEG_TYPE;
            16#F7CB:
                Type	:= '8F1I01.AB2B.0000-1';
                Length	:= 0.450585;
                Valid := 1;
            16#F7CC:
                Type	:= '8F1I01.BA2B.0000-1';
                Length	:= 0.450585;
                Valid := 1;
            ELSE
                Type	:= 'unknown';
                Length	:= 0.0;
                Error := 1;
                ErrorID := ERR_INVALID_SEG_TYPE;
        END_CASE
    ELSE
        Error := 0;
        ErrorID := ERR_OK;
        Valid := 0;
        Type := '';
        Length := 0.0;
    END_IF

END_FUNCTION_BLOCK
```

### Program Logical/Source/Vis (IEC) - Scene viewer interface task

#### Types.typ
```iecst
TYPE
	UserVisTyp : 	STRUCT
		Vis : {REDUND_UNREPLICABLE} McAcpTrakAssemblyVisData;
		Star1RotZ : REAL;
		Star2RotZ : REAL;
	END_STRUCT;
	gUserDataType : 	STRUCT  (*Shuttle User Data*)
		Color : gShuttleColorEnum; (*Shuttle color*)
	END_STRUCT;
	gShuttleColorEnum :
		( (*Shuttle color*)
		SHUTTLE_COLOR_WHITE, (*White shuttles*)
		SHUTTLE_COLOR_BLACK, (*Black shuttles*)
		SHUTTLE_COLOR_GRAY, (*Gray shuttles*)
		SHUTTLE_COLOR_RED, (*Red shuttles*)
		SHUTTLE_COLOR_GREEN, (*Green shuttles*)
		SHUTTLE_COLOR_BLUE, (*Blue shuttles*)
		SHUTTLE_COLOR_YELLOW, (*Yellow shuttles*)
		SHUTTLE_COLOR_PINK, (*Pink shuttles*)
		SHUTTLE_COLOR_ORANGE, (*Orange shuttles*)
		SHUTTLE_COLOR_PURPLE (*Purple shuttles*)
		);
END_TYPE
```

#### Variables.var
```iecst
VAR
	pUserData : REFERENCE TO gUserDataType;
	Vis : McAcpTrakAssemblyVisData;
	SizeofVis : UDINT := 0;
	NumVisShuttle : USINT := 0;
	i : USINT := 0;
	UserVis : {REDUND_UNREPLICABLE} UserVisTyp;
	MC_ReadActualPosInfeed : MC_ReadActualPosition;
	MC_ReadActualPosOutfeed : MC_ReadActualPosition;
	InfeedMasterPos : LREAL;
	OutfeedMasterPos : LREAL;
	plcSimulated : BOOL;
	DiagUserDataAddress : UDINT;
	DiagReadUserData : BOOL;
	DiagUserData : gUserDataType;
	ShuttleMon : McAcpTrakAssemblyMonData; (*Shuttle monitor interface used for scene viewer*)
END_VAR
```

#### Main.st
```iecst
PROGRAM _INIT

	// size of Vis structure - this value has to be entered in B&R scene viewer (PVI -> Options -> Size)
	SizeofVis := SIZEOF(Vis);
	// max number of displayed shuttles
	NumVisShuttle := SIZEOF(Vis.Shuttle) / SIZEOF(Vis.Shuttle[0]);
	// determine if CPU is simulated
	plcSimulated := DiagCpuIsSimulated();

END_PROGRAM

PROGRAM _CYCLIC

	// Simple diagnostic tool to read shuttle user data
	IF EDGEPOS(DiagReadUserData) THEN
		brsmemcpy(ADR(DiagUserData), DiagUserDataAddress, SIZEOF(DiagUserData));
	END_IF

	FOR i := 0 TO (NumVisShuttle - 1) DO
		IF ShuttleMon.Shuttle[i].Available THEN
			// format selected monitor data to fit B&R scene viewer
			Vis.Shuttle[i].Available    := 1;
			Vis.Shuttle[i].PositionX    := LREAL_TO_REAL(ShuttleMon.Shuttle[i].Position.X);
			Vis.Shuttle[i].PositionY    := LREAL_TO_REAL(ShuttleMon.Shuttle[i].Position.Y);
			Vis.Shuttle[i].RotationZ    := LREAL_TO_REAL(ShuttleMon.Shuttle[i].Orientation.Angle1);
			Vis.Shuttle[i].ExtentToFront    := LREAL_TO_REAL(ShuttleMon.Shuttle[i].ExtentToFront);
			Vis.Shuttle[i].ExtentToBack        := LREAL_TO_REAL(ShuttleMon.Shuttle[i].ExtentToBack);
			Vis.Shuttle[i].Width    := LREAL_TO_REAL(ShuttleMon.Shuttle[i].Width);
			IF NOT plcSimulated THEN
				brsitoa(ShuttleMon.Shuttle[i].Index, ADR(Vis.Shuttle[i].Text));
			END_IF

			Vis.Shuttle[i].ColorRed    := 0.5;    //
			Vis.Shuttle[i].ColorGreen    := 0.5;    // default shuttle color grey
			Vis.Shuttle[i].ColorBlue    := 0.5;        //

			IF ShuttleMon.Shuttle[i].UserData <> 0 THEN
				pUserData ACCESS ShuttleMon.Shuttle[i].UserData;
//				IF plcSimulated THEN //Overwrite the Shuttle ID from the ShuttleMon Index with the ID that is in the Userdata to assist in troubleshooting
//					brsitoa(pUserData.ShuttleID, ADR(Vis.Shuttle[i].Text));
//				END_IF

                CASE pUserData.Color OF

                    SHUTTLE_COLOR_GRAY:

                        Vis.Shuttle[i].ColorRed := 0.5;
                        Vis.Shuttle[i].ColorGreen := 0.5;
                        Vis.Shuttle[i].ColorBlue := 0.5;

                    SHUTTLE_COLOR_WHITE:

                        Vis.Shuttle[i].ColorRed := 1.0;
                        Vis.Shuttle[i].ColorGreen := 1.0;
                        Vis.Shuttle[i].ColorBlue := 1.0;

                    SHUTTLE_COLOR_BLACK:

                        Vis.Shuttle[i].ColorRed := 0.0;
                        Vis.Shuttle[i].ColorGreen := 0.0;
                        Vis.Shuttle[i].ColorBlue := 0.0;

                    SHUTTLE_COLOR_RED:

    					Vis.Shuttle[i].ColorRed := 1.0;
    					Vis.Shuttle[i].ColorGreen := 0.0;
                        Vis.Shuttle[i].ColorBlue := 0.0;

                    SHUTTLE_COLOR_PINK:

                        Vis.Shuttle[i].ColorRed := 1.0;
                        Vis.Shuttle[i].ColorGreen := 0.25;
                        Vis.Shuttle[i].ColorBlue := 0.5;

                    SHUTTLE_COLOR_GREEN:

    					Vis.Shuttle[i].ColorRed := 0.0;
    					Vis.Shuttle[i].ColorGreen := 1.0;
    					Vis.Shuttle[i].ColorBlue := 0.0;

    			    SHUTTLE_COLOR_BLUE:
    					Vis.Shuttle[i].ColorRed := 0.0;
    					Vis.Shuttle[i].ColorGreen := 0.0;
    					Vis.Shuttle[i].ColorBlue := 1.0;

    				SHUTTLE_COLOR_YELLOW:
    					Vis.Shuttle[i].ColorRed := 0.8;
    					Vis.Shuttle[i].ColorGreen := 0.8;
    					Vis.Shuttle[i].ColorBlue := 0.0;

    				SHUTTLE_COLOR_ORANGE:
    					Vis.Shuttle[i].ColorRed := 1.0;
    					Vis.Shuttle[i].ColorGreen := 0.5;
                        Vis.Shuttle[i].ColorBlue := 0.0;

                    SHUTTLE_COLOR_PURPLE:
                        Vis.Shuttle[i].ColorRed := 0.6;
                        Vis.Shuttle[i].ColorGreen := 0.0;
                        Vis.Shuttle[i].ColorBlue := 1.0;

                    ELSE

    					Vis.Shuttle[i].ColorRed := 0.5;
    					Vis.Shuttle[i].ColorGreen := 0.5;
                        Vis.Shuttle[i].ColorBlue := 0.5;

                END_CASE

			END_IF
		ELSE
			brsmemset(ADR(Vis.Shuttle[i]), 0, SIZEOF(Vis.Shuttle[0]));
		END_IF
	END_FOR

	UserVis.Vis := Vis;

END_PROGRAM
```

- gMcAssembly01.wsp (not shown)

Listed in the project but not available here: Logical/Global.typ, Logical/Global.var, Logical/Source/Diagnostic/Maint/Exit.st, Logical/Report
